FUNCTION SwapNums
VAR_IN_OUT
	nNumber1 : INT;
	nNumber2 : INT;
END_VAR
VAR
	nNumberTemp : INT;
END_VAR

nNumberTemp := nNumber1;
nNumber1 := nNumber2;
nNumber2 := nNumberTemp;

END_FUNCTION

(* stored: Version 1.1.0.1, ProductVersion 3.1.4024.11
   POU SwapNums: Id {b59f6234-608f-4d78-b6c4-61d6ef3fc1b8}, SpecialFunc None *)
